// TIA Portal project "2" (V15)
// Vorlageprojekt für das Buch mit Zielsystem S7-1200

(* hardware
DEVICE "S7-1200-Station_1"  S7-1200 Station
   slot 0: "Baugruppenträger_0"  Rack  V1.0
   slot 1: "PLC_1"  CPU 1211C DC/DC/DC  6ES7 211-1AE40-0XB0  V4.1
*)

// ===== PLC "PLC_1"  CPU 1211C DC/DC/DC =====

VAR_GLOBAL   // PLC tag table "Standard-Variablentabelle"
   "x" AT %M0.0 : Bool;
   "start" AT %I10.0 : Bool;
   "stop" AT %I10.1 : Bool;
   "C" AT %Q10.0 : Bool;
   "BACK" AT %I10.4 : Bool;
   "pusher" AT %Q10.1 : Bool;
   "FRONT" AT %I10.5 : Bool;
   "SMALL" AT %I10.2 : Bool;
   "Tag_1" AT %M0.1 : Bool;
   "large" AT %I10.3 : Bool;
   "Tag_2" AT %M0.2 : Bool;
   "Tag_3" AT %M0.3 : Bool;
END_VAR

FUNCTION "MHJ-PLC-Lab-Function-S71200" : Void   // FC9000, SCL
{ S7_Optimized_Access := 'TRUE' }
VERSION : 0.1
   VAR_TEMP
      rdTimeReturn : Int;
      outputTime : DTL;
      SyncVal : Byte;
      forVal : Int;
      forVal_2 : Int;
      Value : Byte;
   END_VAR
   VAR CONSTANT
      CompVal : Byte := 16#34;
      Value_01 : Byte := 16#11;
      Value_01_DW : DWord := 16#A165_D992;
      Value_02_DW : DWord := 16#58BE_4401;
   END_VAR
BEGIN

   #Value:=PEEK(area := 16#82,
        dbNumber := 0,
        byteOffset := 511);
   #Value := #Value + 1;

   POKE(area := 16#82,
        dbNumber := 0,
        byteOffset := 511,
        value := #Value);

   POKE(area:=16#81,
        dbNumber:=0,
        byteOffset:=1016,
        value:=#Value_01_DW);
   POKE(area := 16#81,
        dbNumber := 0,
        byteOffset := 1020,
        value := #Value_02_DW);

   POKE(area := 16#81,
        dbNumber := 0,
        byteOffset := 511,
        value := B#16#00);

   FOR #forVal := 0 TO 120 DO
       FOR #forVal_2:=0 TO 10 DO
           #rdTimeReturn:=RD_SYS_T(#outputTime);
           #rdTimeReturn := WR_SYS_T(#outputTime);
           #rdTimeReturn := RD_SYS_T(#outputTime);
           #rdTimeReturn := WR_SYS_T(#outputTime);
       END_FOR;
       #SyncVal:= PEEK(area := 16#81,
                      dbNumber := 0,
                      byteOffset := 511);
       IF #SyncVal = #CompVal THEN
          GOTO M_1;
       END_IF;
   END_FOR;
   RETURN;

   M_1:
   POKE(area := 16#81,
        dbNumber := 0,
        byteOffset := 511,
        value := B#16#0);
END_FUNCTION

ORGANIZATION_BLOCK "Main"   // OB1, LAD, ProgramCycle
TITLE = "Main Program Sweep (Cycle)"
{ S7_Optimized_Access := 'TRUE' }
VERSION : 0.1
   VAR_INPUT
      Initial_Call : Bool;   // Initial call of this OB
      Remanence : Bool;   // =True, if remanent data are available
   END_VAR
BEGIN

REGION Network 1: Konnektierungsbaustein für PLC-Lab
   // Im Netzwerk 1 wird der Konnektierungsbaustein für PLC-Lab aufgerufen.
   // Dieser Aufruf darf nicht entfernt werden!
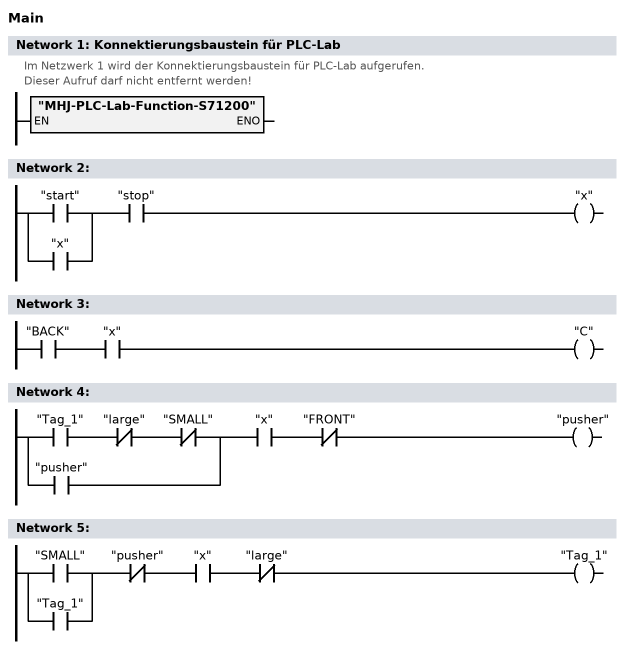
   RUNG wire#powerrail
      "MHJ-PLC-Lab-Function-S71200"()
   END_RUNG
   // the same network as SCL:
   "MHJ-PLC-Lab-Function-S71200"();
END_REGION

REGION Network 2
   RUNG wire#powerrail
      Contact( "start" )
      wire#w1
      Contact( "stop" )
      Coil( "x" )
   END_RUNG
   RUNG wire#powerrail
      Contact( "x" )
   END_RUNG wire#w1
   // the same network as SCL:
   "x" := ("start" OR "x") AND "stop";
END_REGION

REGION Network 3
   RUNG wire#powerrail
      Contact( "BACK" )
      Contact( "x" )
      Coil( "C" )
   END_RUNG
   // the same network as SCL:
   "C" := "BACK" AND "x";
END_REGION

REGION Network 4
   RUNG wire#powerrail
      Contact( "Tag_1" )
      I_Contact( "large" )
      I_Contact( "SMALL" )
      wire#w1
      Contact( "x" )
      I_Contact( "FRONT" )
      Coil( "pusher" )
   END_RUNG
   RUNG wire#powerrail
      Contact( "pusher" )
   END_RUNG wire#w1
   // the same network as SCL:
   "pusher" := (("Tag_1" AND NOT "large" AND NOT "SMALL") OR "pusher") AND "x" AND NOT "FRONT";
END_REGION

REGION Network 5
   RUNG wire#powerrail
      Contact( "SMALL" )
      wire#w1
      I_Contact( "pusher" )
      Contact( "x" )
      I_Contact( "large" )
      Coil( "Tag_1" )
   END_RUNG
   RUNG wire#powerrail
      Contact( "Tag_1" )
   END_RUNG wire#w1
   // the same network as SCL:
   "Tag_1" := ("SMALL" OR "Tag_1") AND NOT "pusher" AND "x" AND NOT "large";
END_REGION
END_ORGANIZATION_BLOCK